// TwinCAT 3 PLC project Lectures
// ProgramVersion: 3.1.4024.0
// libraries:
//   Tc2_Standard, * (Beckhoff Automation GmbH)
//   Tc2_System, * (Beckhoff Automation GmbH)
//   Tc3_Module, * (Beckhoff Automation GmbH)
// project tree:
//   DUTs/ Item.TcDUT, Location.TcDUT (not stored)
//   GVLs/ Automatic.TcGVL, IO.TcGVL (not stored)
//   / PlcTask.TcTTO (not stored)
//   POUs/ AutomaticControl.TcPOU, CountCurrentPosition1.TcPOU, Initialize.TcPOU (not stored), ManualControl.TcPOU, MAIN.TcPOU, MotorSelection.TcPOU, Recipe1.TcPOU, Recipe11.TcPOU, Recipe2.TcPOU, RestorePreviousAutomaticState.TcPOU, Safety1.TcPOU
//   POUs/Lectures%27 programs/ p00_true_false.TcPOU (not stored), p01_sequential.TcPOU (not stored), p02_clock.TcPOU (not stored), p03_SR1.TcPOU (not stored), p04_latch.TcPOU (not stored), p05_posEdge.TcPOU (not stored), p06_frontDetection.TcPOU (not stored), p07_memoryCell.TcPOU (not stored), p08_counter.TcPOU (not stored), p09_timers.TcPOU (not stored), p10_directionalInterlock.TcPOU (not stored), p11_logicalFunction.TcPOU (not stored), p12_controlLight.TcPOU (not stored)
// real-time tasks:
//   TASK PlcTask1: cycle T#10ms, priority 21, ADS port 351
//   TASK PlcTask: cycle T#10ms, priority 20, ADS port 350
// I/O:
//   DEVICE Device 1 (EtherCAT), AmsNetId 172.31.192.1.2.1
//     Term 1 (EK1200) [EK1200-7000 EtherCAT Power supply (1,5A E-Bus)]
//       Term 2 (EL1859) [EL1859 8Ch. Dig. Input 24V, 3ms, 8Ch. Dig. Output 24V, 0.5A]
//       Term 3 (EL1859) [EL1859 8Ch. Dig. Input 24V, 3ms, 8Ch. Dig. Output 24V, 0.5A]
//       Term 4 (EL9011) [EL9011 End Terminal]
//   DEVICE Device 2 (NOV-DP-RAM) (disabled)
//   DEVICE Device 3 (CX7000), AmsNetId 172.31.192.1.4.1
//     Term 1 (CX7028) [CX7028-0000-0121]
//       modules: Module 1 (DIO_2x), Module 2 (Empty Module), Module 3 (DIO_2x), Module 4 (Empty Module), Module 5 (DI_2x), Module 6 (Empty Module), Module 7 (DI_2x), Module 8 (Empty Module)
// variable links:
//   Lectures/Lectures Instance <-> Device 1 (EtherCAT)/Term 1 (EK1200)/Term 2 (EL1859)
//     PlcTask Inputs/IO.EndExtensionSensor <-> Channel 3/Input
//     PlcTask Inputs/IO.EndGripSensor <-> Channel 7/Input
//     PlcTask Inputs/IO.EndLiftingSensor <-> Channel 5/Input
//     PlcTask Inputs/IO.EndRotationSensor <-> Channel 1/Input
//     PlcTask Inputs/IO.StepExtensionSwitch <-> Channel 4/Input
//     PlcTask Inputs/IO.StepGripSwitch <-> Channel 8/Input
//     PlcTask Inputs/IO.StepLiftingSwitch <-> Channel 6/Input
//     PlcTask Inputs/IO.StepRotatonSwitch <-> Channel 2/Input
//     PlcTask Outputs/IO.MotorExtension <-> Channel 12/Output
//     PlcTask Outputs/IO.MotorExtensionDirection <-> Channel 11/Output
//     PlcTask Outputs/IO.MotorGrip <-> Channel 16/Output
//     PlcTask Outputs/IO.MotorGripDirection <-> Channel 15/Output
//     PlcTask Outputs/IO.MotorLifting <-> Channel 14/Output
//     PlcTask Outputs/IO.MotorLiftingDirection <-> Channel 13/Output
//     PlcTask Outputs/IO.MotorRotation <-> Channel 10/Output
//     PlcTask Outputs/IO.MotorRotationDirection <-> Channel 9/Output
//   Lectures/Lectures Instance <-> Device 3 (CX7000)/Term 1 (CX7028)
//     PlcTask Inputs/IO.ButtonGreen <-> Module 3 (DIO_2x)/DIO_2x Input Channel 2/Input
//     PlcTask Inputs/IO.ButtonLowerLeft <-> Module 5 (DI_2x)/DI_2x Input Channel 1/Input
//     PlcTask Inputs/IO.ButtonLowerRight <-> Module 5 (DI_2x)/DI_2x Input Channel 2/Input
//     PlcTask Inputs/IO.ButtonRed <-> Module 1 (DIO_2x)/DIO_2x Input Channel 1/Input
//     PlcTask Inputs/IO.ButtonUpperLeft <-> Module 1 (DIO_2x)/DIO_2x Input Channel 2/Input
//     PlcTask Inputs/IO.ButtonUpperRight <-> Module 3 (DIO_2x)/DIO_2x Input Channel 1/Input
//     PlcTask Inputs/IO.Switch <-> Module 7 (DI_2x)/DI_2x Input Channel 1/Input
//     PlcTask Outputs/IO.LEDBlueLower <-> Module 3 (DIO_2x)/DIO_2x Output Channel 2/Output
//     PlcTask Outputs/IO.LEDBlueUpper <-> Module 1 (DIO_2x)/DIO_2x Output Channel 2/Output
//     PlcTask Outputs/IO.LEDGreen <-> Module 3 (DIO_2x)/DIO_2x Output Channel 1/Output
//     PlcTask Outputs/IO.LEDRed <-> Module 1 (DIO_2x)/DIO_2x Output Channel 1/Output

// ---- DUTs/Item.TcDUT
TYPE Item :
STRUCT
END_STRUCT
END_TYPE

// ---- GVLs/Automatic.TcGVL
{attribute 'qualified_only'}
VAR_GLOBAL
	RCurrentlyMoving: BOOL;
	RotationPositionAuto: INT;
	RotationPositionCurrent: INT;
	SafetyRON: BOOL;
	
	LCurrentlyMoving: BOOL;
	LiftingPositionAuto: INT;
	LiftingPositionCurrent: INT;
	SafetyLON: BOOL;
	
	ECurrentlyMoving: BOOL;
	ExtensionPositionAuto: INT;
	ExtensionPositionCurrent: INT;
	SafetyEON: BOOL;
	
	GCurrentlyMoving: BOOL;
	GripPositionAuto: INT;
	GripPositionCurrent: INT;
	SafetyGON: BOOL;
	
	AllRestored: BOOL;
END_VAR

// ---- POUs/AutomaticControl.TcPOU
FUNCTION_BLOCK PUBLIC AutomaticControl
VAR_INPUT
    Switch: BOOL;
END_VAR
VAR
    State: INT := 0;
    ExecutingRecipe1: BOOL := FALSE;
    ExecutingRecipe2: BOOL := FALSE;
	myRecipe1: Recipe1;
    myRecipe2: Recipe2;
    Tmp: BOOL;
    RestorePreviousAutomaticState: RestorePreviousAutomaticState;
	CountCurrentPosition1: CountCurrentPosition1;
	Safety: Safety1;
END_VAR
VAR_OUTPUT
    Output: BOOL := TRUE;
END_VAR

// TwinCAT ensures that all POUs, including your AutomaticControl program 
// and Recipe1() Function Block, are executed once per cycle.

// for debugging purposes:
IF IO.ButtonRed THEN
	IO.Initialized := FALSE;
END_IF


IF (NOT IO.Initialized) THEN
	Initialize();
ELSIF (NOT IO.Switch) AND IO.PreviousManualMode THEN
	CountCurrentPosition1();
	Safety();
	RestorePreviousAutomaticState();
ELSE
	CountCurrentPosition1();
	Safety();
	
    IF (IO.ButtonUpperLeft OR ExecutingRecipe1) AND Automatic.AllRestored THEN
        //ExecutingRecipe1 := TRUE;
		//Recipe11();
        //ExecutingRecipe1 := NOT Recipe11.SuccesfullyEnded; // Update ExecutingRecipe1 based on output
		myRecipe1.ExecutingRecipe1 := TRUE;
		ExecutingRecipe1 := NOT myRecipe1.SuccesfullyEnded;
    ELSIF (NOT ExecutingRecipe1) AND (IO.ButtonUpperRight OR ExecutingRecipe2) AND Automatic.AllRestored THEN
        ExecutingRecipe2 := TRUE;
        myRecipe2.ExecutingRecipe2 := ExecutingRecipe2; // Pass input to the function block
        //myRecipe2(); // Call the function block
        ExecutingRecipe2 := NOT myRecipe2.SuccesfullyEnded; // Update ExecutingRecipe2 based on output
    END_IF
END_IF




RETURN;

END_FUNCTION_BLOCK

// ---- POUs/Recipe1.TcPOU
FUNCTION_BLOCK Recipe1
VAR_INPUT
	ExecutingRecipe1: BOOL;
END_VAR
VAR_OUTPUT
	SuccesfullyEnded: BOOL := FALSE;
END_VAR
VAR
	State: INT := 0;
	WoodInitialLiftingPosition: INT := 50;
	InitialExtensionPosition: INT := 388;
	MaxGripPosition: INT := 150;
	RotationDropOffPosition: INT := 300;
	PlasticsInitialLiftingPosition: INT := 250;
	PlasticsDropOffExtensionPosition: INT := 300;
	MetalInitialLiftingPosition: INT := 400;
	MetalDropOffExtensionPosition: INT := 500;
END_VAR

IF ExecutingRecipe1 THEN	// we start executing recipe1 (again)
	SuccesfullyEnded := FALSE;
END_IF

IF (NOT IO.Switch) AND (NOT SuccesfullyEnded) THEN
	IO.LEDGreen := 1;
	// WOOD:
	IF State = 0 THEN
		IF Automatic.LiftingPositionAuto < WoodInitialLiftingPosition THEN
			IO.MotorLiftingDirection := 0;
			IF (NOT Automatic.SafetyLON) THEN
				Automatic.LCurrentlyMoving := TRUE;
				IO.MotorLifting := 1;
			END_IF
		ELSE
			State := 1;
			IO.MotorLifting := 0;
			Automatic.LCurrentlyMoving := FALSE;
		END_IF
	ELSIF State = 1 THEN
		IF Automatic.ExtensionPositionAuto < InitialExtensionPosition THEN
			IO.MotorExtensionDirection := 0;
			IF NOT Automatic.SafetyEON THEN
				Automatic.ECurrentlyMoving := TRUE;
				IO.MotorExtension := 1;
			END_IF
		ELSE
			State := 2;
			IO.MotorExtension := 0;
			Automatic.ECurrentlyMoving := FALSE;
		END_IF
	ELSIF State = 2 THEN
		IF Automatic.GripPositionAuto < MaxGripPosition THEN
			IO.MotorGripDirection := 0;
			IF NOT Automatic.SafetyGON THEN
				Automatic.GCurrentlyMoving := TRUE;
				IO.MotorGrip := 1;
			END_IF
		ELSE
			State := 3;
			IO.MotorGrip := 0;
			Automatic.GCurrentlyMoving := FALSE;
		END_IF
	ELSIF State = 3 THEN
		IF NOT IO.EndLiftingSensor THEN
			IO.MotorLiftingDirection := 1;
			IF NOT Automatic.SafetyLON THEN
				Automatic.GCurrentlyMoving := TRUE;
				IO.MotorLifting := 1;
			END_IF
		ELSE
			State := 4;
			IO.MotorLifting := 0;
			Automatic.LCurrentlyMoving := FALSE;
		END_IF
	ELSIF State = 4 THEN
		IF Automatic.RotationPositionAuto < RotationDropOffPosition THEN
			IO.MotorRotationDirection := 0;
			IF NOT Automatic.SafetyRON THEN
				Automatic.RCurrentlyMoving := TRUE;
				IO.MotorRotation := 1;
			END_IF
		ELSE
			State := 5;
			IO.MotorRotation := 0;
			Automatic.RCurrentlyMoving := FALSE;
		END_IF
	ELSIF State = 5 THEN
		IF NOT IO.EndExtensionSensor THEN	// it drops wood in the nearest bin
			IO.MotorExtensionDirection := 1;
			IF NOT Automatic.SafetyEON THEN
				Automatic.ECurrentlyMoving := TRUE;
				IO.MotorExtension := 1;
			END_IF
		ELSE
			State := 6;
			IO.MotorExtension := 0;
			Automatic.ECurrentlyMoving := FALSE;
		END_IF
	ELSIF State = 6 THEN
		IF NOT IO.EndGripSensor THEN
			IO.MotorGripDirection := 1;
			IF NOT Automatic.SafetyGON THEN
				Automatic.GCurrentlyMoving := TRUE;
				IO.MotorGrip := 1;
			END_IF
		ELSE
			State := 7;
			IO.MotorGrip := 0;
			Automatic.GCurrentlyMoving := FALSE;
		END_IF
	ELSIF State = 7 THEN
		IF NOT IO.EndRotationSensor THEN
			IO.MotorRotationDirection := 1;
			IF NOT Automatic.SafetyRON THEN
				Automatic.RCurrentlyMoving := TRUE;
				IO.MotorRotation := 1;
			END_IF
		ELSE
			State := 8;
			IO.MotorRotation := 0;
			Automatic.RCurrentlyMoving := FALSE;
		END_IF
	END_IF
	
	// PLASTICS:
	IF State = 8 THEN
		IF Automatic.LiftingPositionAuto < PlasticsInitialLiftingPosition THEN
			IO.MotorLiftingDirection := 0;
			IF NOT Automatic.SafetyLON THEN
				Automatic.LCurrentlyMoving := TRUE;
				IO.MotorLifting := 1;
			END_IF
		ELSE
			State := 9;
			IO.MotorLifting := 0;
			Automatic.LCurrentlyMoving := FALSE;
		END_IF
	ELSIF State = 9 THEN
		IF Automatic.ExtensionPositionAuto < InitialExtensionPosition THEN
			IO.MotorExtensionDirection := 0;
			IF NOT Automatic.SafetyEON THEN
				Automatic.ECurrentlyMoving := TRUE;
				IO.MotorExtension := 1;
			END_IF
		ELSE
			State := 10;
			IO.MotorExtension := 0;
			Automatic.ECurrentlyMoving := FALSE;
		END_IF
	ELSIF State = 10 THEN
		IF Automatic.GripPositionAuto < MaxGripPosition THEN
			IO.MotorGripDirection := 0;
			IF NOT Automatic.SafetyGON THEN
				Automatic.GCurrentlyMoving := TRUE;
				IO.MotorGrip := 1;
			END_IF
		ELSE
			State := 11;
			IO.MotorGrip := 0;
			Automatic.GCurrentlyMoving := FALSE;
		END_IF
	ELSIF State = 11 THEN
		IF NOT IO.EndLiftingSensor THEN
			IO.MotorLiftingDirection := 1;
			IF NOT Automatic.SafetyLON THEN
				Automatic.LCurrentlyMoving := TRUE;
				IO.MotorLifting := 1;
			END_IF
		ELSE
			State := 12;
			IO.MotorLifting := 0;
			Automatic.LCurrentlyMoving := FALSE;
		END_IF
	ELSIF State = 12 THEN
		IF Automatic.RotationPositionAuto < RotationDropOffPosition THEN
			IO.MotorRotationDirection := 0;
			IF NOT Automatic.SafetyRON THEN
				Automatic.RCurrentlyMoving := TRUE;
				IO.MotorRotation := 1;
			END_IF
		ELSE
			State := 13;
			IO.MotorRotation := 0;
			Automatic.RCurrentlyMoving := FALSE;
		END_IF
	ELSIF State = 13 THEN
		IF Automatic.ExtensionPositionAuto > PlasticsDropOffExtensionPosition THEN	// it drops plastics into second nearest bin
			IO.MotorExtensionDirection := 1;
			IF NOT Automatic.SafetyEON THEN
				Automatic.ECurrentlyMoving := TRUE;
				IO.MotorExtension := 1;
			END_IF
		ELSE
			State := 14;
			IO.MotorExtension := 0;
			Automatic.ECurrentlyMoving := FALSE;
		END_IF
	ELSIF State = 14 THEN
		IF NOT IO.EndGripSensor THEN
			IO.MotorGripDirection := 1;
			IF NOT Automatic.SafetyGON THEN
				Automatic.GCurrentlyMoving := TRUE;
				IO.MotorGrip := 1;
			END_IF
		ELSE
			State := 15;
			IO.MotorGrip := 0;
			Automatic.GCurrentlyMoving := FALSE;
		END_IF
	ELSIF State = 15 THEN
		IF NOT IO.EndRotationSensor THEN
			IO.MotorRotationDirection := 0;
			IF NOT Automatic.SafetyRON THEN
				Automatic.RCurrentlyMoving := TRUE;
				IO.MotorRotation := 1;
			END_IF
		ELSE
			State := 16;
			IO.MotorRotation := 0;
			Automatic.RCurrentlyMoving := FALSE;
		END_IF
	END_IF
	
	// METAL:
	IF State = 16 THEN
		IF Automatic.LiftingPositionAuto < MetalInitialLiftingPosition THEN
			IO.MotorLiftingDirection := 0;
			IF NOT Automatic.SafetyLON THEN
				Automatic.LCurrentlyMoving := TRUE;
				IO.MotorLifting := 1;
			END_IF
		ELSE
			State := 17;
			IO.MotorLifting := 0;
			Automatic.LCurrentlyMoving := FALSE;
		END_IF
	ELSIF State = 17 THEN
		IF Automatic.ExtensionPositionAuto < InitialExtensionPosition THEN
			IO.MotorExtensionDirection := 0;
			IF NOT Automatic.SafetyEON THEN
				Automatic.ECurrentlyMoving := TRUE;
				IO.MotorExtension := 1;
			END_IF
		ELSE
			State := 18;
			IO.MotorExtension := 0;
			Automatic.ECurrentlyMoving := FALSE;
		END_IF
	ELSIF State = 18 THEN
		IF Automatic.GripPositionAuto < MaxGripPosition THEN
			IO.MotorGripDirection := 0;
			IF NOT Automatic.SafetyGON THEN
				Automatic.GCurrentlyMoving := TRUE;
				IO.MotorGrip := 1;
			END_IF
		ELSE
			State := 19;
			IO.MotorGrip := 0;
			Automatic.GCurrentlyMoving := FALSE;
		END_IF
	ELSIF State = 19 THEN
		IF NOT IO.EndLiftingSensor THEN
			IO.MotorLiftingDirection := 1;
			IF NOT Automatic.SafetyLON THEN
				Automatic.LCurrentlyMoving := TRUE;
				IO.MotorLifting := 1;
			END_IF
		ELSE
			State := 20;
			IO.MotorLifting := 0;
			Automatic.LCurrentlyMoving := FALSE;
		END_IF
	ELSIF State = 20 THEN
		IF Automatic.RotationPositionAuto < RotationDropOffPosition THEN
			IO.MotorRotationDirection := 0;
			IF NOT Automatic.SafetyRON THEN
				Automatic.RCurrentlyMoving := TRUE;
				IO.MotorRotation := 1;
			END_IF
		ELSE
			State := 21;
			IO.MotorRotation := 0;
			Automatic.RCurrentlyMoving := FALSE;
		END_IF
	ELSIF State = 21 THEN
		IF Automatic.ExtensionPositionAuto > MetalDropOffExtensionPosition THEN	// it drops metal into farthest bin
			IO.MotorExtensionDirection := 1;
			IF NOT Automatic.SafetyEON THEN
				Automatic.ECurrentlyMoving := TRUE;
				IO.MotorExtension := 1;
			END_IF
		ELSE
			State := 22;
			IO.MotorExtension := 0;
			Automatic.ECurrentlyMoving := FALSE;
		END_IF
	ELSIF State = 22 THEN
		IF NOT IO.EndGripSensor THEN
			IO.MotorGripDirection := 1;
			IF NOT Automatic.SafetyGON THEN
				Automatic.GCurrentlyMoving := TRUE;
				IO.MotorGrip := 1;
			END_IF
		ELSE
			State := 23;
			IO.MotorGrip := 0;
			Automatic.GCurrentlyMoving := FALSE;
		END_IF
	ELSIF State = 23 THEN
		IF NOT IO.EndRotationSensor THEN
			IO.MotorRotationDirection := 1;
			IF NOT Automatic.SafetyRON THEN
				Automatic.RCurrentlyMoving := TRUE;
				IO.MotorRotation := 1;
			END_IF
		ELSE
			State := 24;
			IO.MotorRotation := 0;
			Automatic.RCurrentlyMoving := FALSE;
		END_IF
	ELSIF State = 24 THEN
		SuccesfullyEnded := TRUE;
		State := 0;
		RETURN;
	END_IF
END_IF
RETURN;

END_FUNCTION_BLOCK

// ---- POUs/Recipe2.TcPOU
FUNCTION_BLOCK PUBLIC Recipe2
VAR_INPUT
	ExecutingRecipe2: BOOL;
END_VAR
VAR_OUTPUT
	SuccesfullyEnded: BOOL := FALSE;
END_VAR
VAR
	State: INT := 0;
	InitialRotationPosition: INT := 140;
	InitialLiftingPosition: INT := 200;
	MaxGripPosition: INT := 160;
END_VAR

// Recipe is sequence of moves to execute the task.

IF ExecutingRecipe2 THEN	// we start executing recipe2 (again)
	SuccesfullyEnded := FALSE;
END_IF

IF NOT IO.Switch AND NOT SuccesfullyEnded THEN
	// WOOD:
	IF State = 0 THEN
		IF Automatic.RotationPositionAuto < InitialRotationPosition THEN
			IO.MotorRotationDirection := 0;
			IF NOT Automatic.SafetyRON THEN
				Automatic.RCurrentlyMoving := TRUE;
				IO.MotorRotation := 1;
			END_IF
		ELSE
			State := 1;
			IO.MotorRotation := 0;
			Automatic.RCurrentlyMoving := FALSE;
		END_IF
	ELSIF State = 1 THEN
		IF Automatic.LiftingPositionAuto < InitialLiftingPosition THEN
			IO.MotorLiftingDirection := 1;
			IF NOT Automatic.SafetyLON THEN
				Automatic.LCurrentlyMoving := TRUE;
				IO.MotorLifting := 1;
			END_IF
		ELSE
			State := 2;
			IO.MotorLifting := 0;
			Automatic.LCurrentlyMoving := FALSE;
		END_IF
	ELSIF State = 2 THEN
		IF Automatic.GripPositionAuto < MaxGripPosition THEN
			IO.MotorGripDirection := 0;
			IF NOT Automatic.SafetyGON THEN
				Automatic.GCurrentlyMoving := TRUE;
				IO.MotorGrip := 1;
			END_IF
		ELSE
			State := 3;
			IO.MotorGrip := 0;
			Automatic.GCurrentlyMoving := FALSE;
		END_IF
	ELSIF State = 3 THEN
		IF NOT IO.EndLiftingSensor THEN
			IO.MotorLiftingDirection := 0;
			IF NOT Automatic.SafetyLON THEN
				Automatic.GCurrentlyMoving := TRUE;
				IO.MotorLifting := 1;
			END_IF
		ELSE
			State := 4;
			IO.MotorLifting := 0;
			Automatic.GCurrentlyMoving := FALSE;
		END_IF
	ELSIF State = 4 THEN
		IF NOT IO.EndRotationSensor THEN
			IO.MotorRotationDirection := 1;
			IF NOT Automatic.SafetyRON THEN
				Automatic.RCurrentlyMoving := TRUE;
				IO.MotorRotation := 1;
			END_IF
		ELSE
			State := 5;
			IO.MotorRotation := 0;
			Automatic.RCurrentlyMoving := FALSE;
		END_IF
	ELSIF State = 5 THEN
		IF NOT IO.EndGripSensor THEN		// it places the cylinder onto the platform
			IO.MotorGripDirection := 1;
			IF NOT Automatic.SafetyGON THEN
				Automatic.GCurrentlyMoving := TRUE;
				IO.MotorGrip := 1;
			END_IF
		ELSE
			State := 6;
			IO.MotorGrip := 0;
			Automatic.GCurrentlyMoving := FALSE;
		END_IF
	ELSIF State = 6 THEN
		SuccesfullyEnded := TRUE;
		State := 0;
		RETURN;
	END_IF
END_IF

END_FUNCTION_BLOCK

// ---- POUs/RestorePreviousAutomaticState.TcPOU
FUNCTION_BLOCK PUBLIC RestorePreviousAutomaticState
VAR_INPUT
END_VAR
VAR_OUTPUT
END_VAR
VAR
	RotationRestored: BOOL := FALSE;
	LiftingRestored: BOOL := FALSE;
	ExtensionRestored: BOOL := FALSE;
	GripRestored: BOOL := FALSE;
END_VAR

IF IO.PreviousManualMode THEN
	Automatic.AllRestored := FALSE;
END_IF

// reset rotation:
IF Automatic.RotationPositionAuto - Automatic.RotationPositionCurrent > 5 AND (NOT RotationRestored) AND (NOT Automatic.SafetyRON) THEN
	IO.MotorRotationDirection := 0;
	Automatic.RCurrentlyMoving := TRUE;
	IO.MotorRotation := 1;
ELSIF Automatic.RotationPositionCurrent - Automatic.RotationPositionAuto > 5 AND (NOT RotationRestored) AND (NOT Automatic.SafetyRON) THEN
	IO.MotorRotationDirection := 1;
	Automatic.RCurrentlyMoving := TRUE;
	IO.MotorRotation := 1;
ELSE
	Automatic.RCurrentlyMoving := FALSE;
	IO.MotorRotation := 0;
	RotationRestored := TRUE;
END_IF

// reset lifting:
IF Automatic.LiftingPositionAuto - Automatic.LiftingPositionCurrent > 5 AND (NOT LiftingRestored) AND (NOT Automatic.SafetyLON) THEN
	IO.MotorLiftingDirection := 0;
	Automatic.LCurrentlyMoving := TRUE;
	IO.MotorLifting := 1;
ELSIF Automatic.LiftingPositionCurrent - Automatic.LiftingPositionAuto > 5 AND (NOT LiftingRestored) AND (NOT Automatic.SafetyLON) THEN
	IO.MotorLiftingDirection := 0;
	Automatic.LCurrentlyMoving := TRUE;
	IO.MotorLifting := 1;
ELSE
	Automatic.LCurrentlyMoving := FALSE;
	IO.MotorLifting := 0;
	LiftingRestored := TRUE;
END_IF

// reset extension:
IF Automatic.ExtensionPositionAuto - Automatic.ExtensionPositionCurrent > 5 AND (NOT ExtensionRestored) AND (NOT Automatic.SafetyEON) THEN
	IO.MotorExtensionDirection := 0;
	Automatic.ECurrentlyMoving := TRUE;
	IO.MotorExtension := 1;
ELSIF Automatic.ExtensionPositionCurrent - Automatic.ExtensionPositionAuto > 5 AND (NOT ExtensionRestored) AND (NOT Automatic.SafetyEON) THEN
	IO.MotorExtensionDirection := 0;
	Automatic.ECurrentlyMoving := TRUE;
	IO.MotorExtension := 1;
ELSE
	Automatic.ECurrentlyMoving := FALSE;
	IO.MotorExtension := 0;
	ExtensionRestored := TRUE;
END_IF

// reset grip:
IF Automatic.GripPositionAuto - Automatic.GripPositionCurrent > 5 AND (NOT GripRestored) AND (NOT Automatic.SafetyGON) THEN
	IO.MotorGripDirection := 0;
	Automatic.GCurrentlyMoving := TRUE;
	IO.MotorGrip := 1;
ELSIF Automatic.GripPositionCurrent - Automatic.GripPositionAuto > 5 AND (NOT GripRestored) AND (NOT Automatic.SafetyGON) THEN
	IO.MotorGripDirection := 0;
	Automatic.GCurrentlyMoving := TRUE;
	IO.MotorGrip := 1;
ELSE
	Automatic.GCurrentlyMoving := FALSE;
	IO.MotorGrip := 0;
	GripRestored := TRUE;
END_IF

// if all restored then go on to exeecute recipes in AutomaticControl:
IF RotationRestored AND LiftingRestored AND ExtensionRestored AND GripRestored THEN
	IO.PreviousManualMode := FALSE;
	Automatic.AllRestored := TRUE;
	
	RotationRestored := FALSE;
	ExtensionRestored := FALSE;
	LiftingRestored := FALSE;
	GripRestored := FALSE;
	Automatic.RCurrentlyMoving := FALSE;
	Automatic.ECurrentlyMoving := FALSE;
	Automatic.LCurrentlyMoving := FALSE;
	Automatic.GCurrentlyMoving := FALSE;
END_IF

END_FUNCTION_BLOCK

// ---- POUs/CountCurrentPosition1.TcPOU
FUNCTION_BLOCK CountCurrentPosition1
VAR_INPUT
END_VAR
VAR_OUTPUT
END_VAR
VAR
END_VAR

IF IO.Initialized THEN
	
	// COUNT ROTATION:
	IF IO.StepRotatonSwitch = 1 AND Automatic.RCurrentlyMoving THEN
		// away from the sensor:
		IF IO.MotorRotationDirection = 0 THEN
			IF (NOT IO.Switch) THEN		// in automatic mode
				IF IO.PreviousManualMode THEN	
					Automatic.RotationPositionCurrent := Automatic.RotationPositionCurrent + 1;
				ELSE	// to restore the state
					Automatic.RotationPositionCurrent := Automatic.RotationPositionCurrent + 1;
					Automatic.RotationPositionAuto := Automatic.RotationPositionAuto + 1;
				END_IF
			ELSE		// in manual mode
				Automatic.RotationPositionCurrent := Automatic.RotationPositionCurrent + 1;
			END_IF
		// towards the sensor:
		ELSE
			IF (NOT IO.Switch) THEN		// in automatic mode
				IF IO.PreviousManualMode THEN	
					Automatic.RotationPositionCurrent := Automatic.RotationPositionCurrent - 1;
				ELSE	// to restore the state
					Automatic.RotationPositionCurrent := Automatic.RotationPositionCurrent - 1;
					Automatic.RotationPositionAuto := Automatic.RotationPositionAuto - 1;
				END_IF
			ELSE		// in manual mode
				Automatic.RotationPositionCurrent := Automatic.RotationPositionCurrent - 1;
			END_IF
		END_IF
	END_IF
	
	// COUNT Extension: (-------edino še NESPREMENJENO--------)
	IF IO.StepExtensionSwitch = 1 THEN
		IF IO.MotorExtensionDirection = 0 THEN
			IF (NOT IO.Switch) AND Automatic.ECurrentlyMoving THEN
				IF IO.PreviousManualMode THEN
					Automatic.ExtensionPositionCurrent := Automatic.ExtensionPositionCurrent + 1;
				ELSE
					Automatic.ExtensionPositionAuto := Automatic.ExtensionPositionAuto + 1;
					Automatic.ExtensionPositionCurrent := Automatic.ExtensionPositionCurrent + 1;
				END_IF
			ELSIF Automatic.ECurrentlyMoving THEN
				Automatic.ExtensionPositionCurrent := Automatic.ExtensionPositionCurrent + 1;
			END_IF
		ELSE
			IF (NOT IO.Switch) AND Automatic.ECurrentlyMoving THEN
				IF IO.PreviousManualMode THEN
					Automatic.ExtensionPositionCurrent := Automatic.ExtensionPositionCurrent - 1;
				ELSE
					Automatic.ExtensionPositionAuto := Automatic.ExtensionPositionAuto - 1;
					Automatic.ExtensionPositionCurrent := Automatic.ExtensionPositionCurrent - 1;
				END_IF
			ELSIF Automatic.ECurrentlyMoving THEN
				Automatic.ExtensionPositionCurrent := Automatic.ExtensionPositionCurrent - 1;
			END_IF
		END_IF
	END_IF
	
	// COUNT Lifting:
	IF IO.StepLiftingSwitch = 1 AND Automatic.LCurrentlyMoving THEN
		// away from the sensor:
		IF IO.MotorLiftingDirection = 0 THEN
			IF (NOT IO.Switch) THEN		// in automatic mode
				IF IO.PreviousManualMode THEN
					Automatic.LiftingPositionCurrent := Automatic.LiftingPositionCurrent + 1;
				ELSE	// to restore the state
					Automatic.LiftingPositionCurrent := Automatic.LiftingPositionCurrent + 1;
					Automatic.LiftingPositionAuto := Automatic.LiftingPositionAuto + 1;
				END_IF
			ELSE		// in manual mode
				Automatic.LiftingPositionCurrent := Automatic.LiftingPositionCurrent + 1;
			END_IF
		// towards the sensor:
		ELSE
			IF (NOT IO.Switch) THEN		// in automatic mode
				IF IO.PreviousManualMode THEN
					Automatic.LiftingPositionCurrent := Automatic.LiftingPositionCurrent - 1;
				ELSE	// to restore the state
					Automatic.LiftingPositionAuto := Automatic.LiftingPositionAuto - 1;
					Automatic.LiftingPositionCurrent := Automatic.LiftingPositionCurrent - 1;
				END_IF
			ELSE		// in manual mode
				Automatic.LiftingPositionCurrent := Automatic.LiftingPositionCurrent - 1;
			END_IF
		END_IF
	END_IF
	
	// COUNT Grip:
	IF IO.StepGripSwitch = 1 AND Automatic.GCurrentlyMoving THEN
		IF IO.MotorGripDirection = 0 THEN
			IF (NOT IO.Switch) THEN		// in automatic mode
				IF IO.PreviousManualMode THEN
					Automatic.GripPositionCurrent := Automatic.GripPositionCurrent + 1;
				ELSE
					Automatic.GripPositionAuto := Automatic.GripPositionAuto + 1;
					Automatic.GripPositionCurrent := Automatic.GripPositionCurrent + 1;
				END_IF
			ELSE		// in manual mode
				Automatic.GripPositionCurrent := Automatic.GripPositionCurrent + 1;
			END_IF
		ELSE
			IF (NOT IO.Switch) THEN		// in automatic mode
				IF IO.PreviousManualMode THEN
					Automatic.GripPositionCurrent := Automatic.GripPositionCurrent - 1;
				ELSE
					Automatic.GripPositionAuto := Automatic.GripPositionAuto - 1;
					Automatic.GripPositionCurrent := Automatic.GripPositionCurrent - 1;
				END_IF
			ELSE		// in manual mode
				Automatic.GripPositionCurrent := Automatic.GripPositionCurrent - 1;
			END_IF
		END_IF
	END_IF
	
END_IF

END_FUNCTION_BLOCK

// ---- POUs/Safety1.TcPOU
FUNCTION_BLOCK Safety1
VAR_INPUT
END_VAR
VAR_OUTPUT
END_VAR
VAR
	MaxRotationPosition: INT := 555;
	MaxLiftingPosition: INT := 270;
	MaxExtensionPosition: INT := 445;
	MaxGripPosition: INT := 155;
END_VAR

// Safety for Rotation:
IF Automatic.RotationPositionCurrent >= MaxRotationPosition AND NOT IO.ButtonLowerLeft AND NOT IO.MotorRotationDirection = 1 THEN
	Automatic.SafetyRON := TRUE;
	IO.MotorRotation := 0;
	IF Automatic.RotationPositionCurrent >= MaxRotationPosition THEN
		Automatic.RotationPositionCurrent := MaxRotationPosition;
	END_IF
	//Automatic.MotorR.CurrentlyMoving := FALSE;
	Automatic.RCurrentlyMoving := FALSE;
END_IF
IF IO.MotorRotationDirection = 0 THEN
	Automatic.SafetyRON := FALSE;
END_IF
IF IO.EndRotationSensor THEN
	IF IO.MotorRotationDirection = 0 THEN
		Automatic.SafetyRON := FALSE;
	ELSE
		Automatic.SafetyRON := TRUE;
		Automatic.RotationPositionCurrent := 0;
		//Automatic.MotorR.CurrentlyMoving := FALSE;
		Automatic.RCurrentlyMoving := FALSE;
	END_IF
END_IF

// Safety for Lifting:
IF Automatic.LiftingPositionCurrent >= MaxLiftingPosition AND NOT IO.ButtonLowerLeft AND NOT IO.MotorLiftingDirection = 1 THEN
	Automatic.SafetyLON := TRUE;
	IO.MotorLifting := 0;
	IF Automatic.LiftingPositionCurrent >= MaxLiftingPosition THEN
		Automatic.LiftingPositionCurrent := MaxLiftingPosition;
	END_IF
	//Automatic.MotorL.CurrentlyMoving := FALSE;
	Automatic.LCurrentlyMoving := FALSE;
END_IF
IF IO.MotorLiftingDirection = 0 THEN
	Automatic.SafetyLON := FALSE;
END_IF
IF IO.EndLiftingSensor THEN
	IF IO.MotorLiftingDirection = 0 THEN
		Automatic.SafetyLON := FALSE;
	ELSE
		Automatic.SafetyLON := TRUE;
		Automatic.LiftingPositionCurrent := 0;
		//Automatic.MotorL.CurrentlyMoving := FALSE;
		Automatic.RCurrentlyMoving := FALSE;
	END_IF
END_IF

// Safety for Extension:
IF Automatic.ExtensionPositionCurrent >= MaxExtensionPosition AND NOT IO.ButtonLowerLeft AND NOT IO.MotorExtensionDirection = 1 THEN
	Automatic.SafetyEON := TRUE;
	IO.MotorExtension := 0;
	IF Automatic.ExtensionPositionCurrent >= MaxExtensionPosition THEN
		Automatic.ExtensionPositionCurrent := MaxExtensionPosition;
	END_IF
	//Automatic.MotorE.CurrentlyMoving := FALSE;
	Automatic.ECurrentlyMoving := FALSE;
END_IF
IF IO.MotorExtensionDirection = 0 THEN
	Automatic.SafetyEON := FALSE;
END_IF
IF IO.EndExtensionSensor THEN
	IF IO.MotorExtensionDirection = 0 THEN
		Automatic.SafetyEON := FALSE;
	ELSE
		Automatic.SafetyEON := TRUE;
		Automatic.ExtensionPositionCurrent := 0;
		//Automatic.MotorE.CurrentlyMoving := FALSE;
		Automatic.ECurrentlyMoving := FALSE;
	END_IF
END_IF

// Safety for Grip:
IF Automatic.GripPositionCurrent >= MaxGripPosition AND NOT IO.ButtonLowerLeft AND IO.MotorGripDirection = 0 THEN
	Automatic.SafetyGON := TRUE;
	IO.MotorGrip := 0;
	IF Automatic.GripPositionCurrent >= MaxGripPosition THEN
		Automatic.GripPositionCurrent := MaxGripPosition;
	END_IF
	//Automatic.GCurrentlyMoving := FALSE;
	Automatic.GCurrentlyMoving := FALSE;
END_IF
IF IO.MotorGripDirection = 1 THEN
	Automatic.SafetyGON := FALSE;
END_IF
IF IO.EndGripSensor THEN
	IF IO.MotorGripDirection = 0 THEN
		Automatic.SafetyGON := FALSE;
	ELSE
		Automatic.SafetyGON := TRUE;
		Automatic.GripPositionCurrent := 0;
		//Automatic.GCurrentlyMoving := FALSE;
		Automatic.GCurrentlyMoving := FALSE;
	END_IF
END_IF

END_FUNCTION_BLOCK

// ---- POUs/ManualControl.TcPOU
FUNCTION_BLOCK PUBLIC ManualControl
VAR_INPUT
	Switch: BOOL;
END_VAR
VAR
	ManualControl: BOOL;
	TimeForInterlockDelay: TIME := T#0.05S;
	ManualMode: BOOL;
	MotorSelection_1: MotorSelection;
	SelectedMotor: INT;
	temp: TIME;
	LowerLeftInterlock: TOF;
	LowerLeft: BOOL;
	LowerRightInterlock: TOF;
	LowerRight: BOOL;
END_VAR
VAR_OUTPUT
	Output: BOOL;
END_VAR
VAR // added by the converter: edge detectors and wires of the graphical bodies
    _w1, _w2, _w3, _w4, _w5, _w6, _w7, _w8, _w9, _w10, _w11 : BOOL;
    _rt1, _rt2, _rt3 : R_TRIG;
    _ft1, _ft2, _ft3 : F_TRIG;
END_VAR

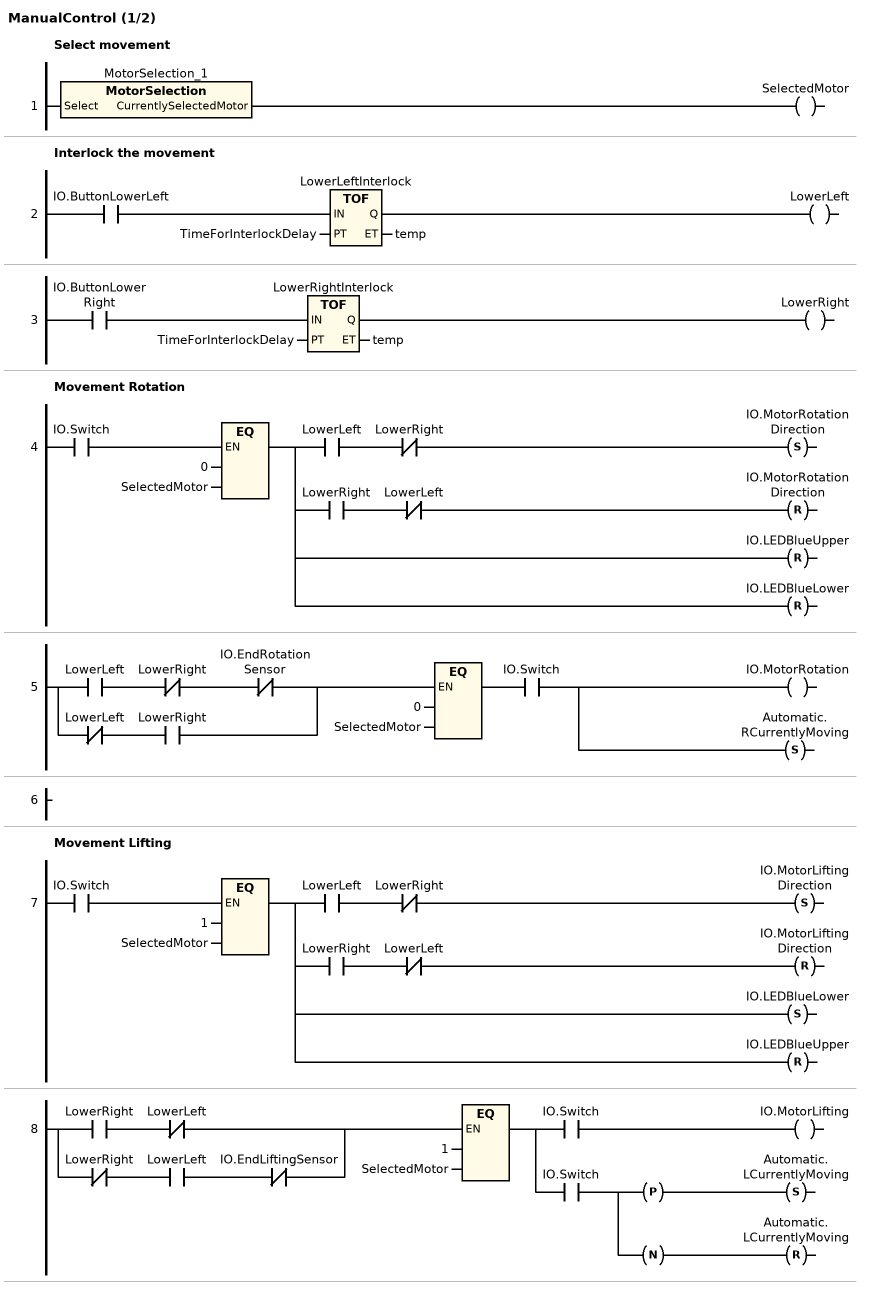
// NETWORK 1: Select movement
MotorSelection_1(Select := TRUE); // MotorSelection
SelectedMotor := MotorSelection_1.CurrentlySelectedMotor;

// NETWORK 2: Interlock the movement
LowerLeftInterlock(IN := IO.ButtonLowerLeft, PT := TimeForInterlockDelay, ET => temp); // TOF
LowerLeft := LowerLeftInterlock.Q;

// NETWORK 3
LowerRightInterlock(IN := IO.ButtonLowerRight, PT := TimeForInterlockDelay, ET => temp); // TOF
LowerRight := LowerRightInterlock.Q;

// NETWORK 4: Movement Rotation
_w1 := IO.Switch AND 0 = SelectedMotor;
IO.MotorRotationDirection S= _w1 AND LowerLeft AND NOT LowerRight;
IO.MotorRotationDirection R= _w1 AND LowerRight AND NOT LowerLeft;
IO.LEDBlueUpper R= _w1;
IO.LEDBlueLower R= _w1;

// NETWORK 5
_w2 := ((LowerLeft AND NOT LowerRight AND NOT IO.EndRotationSensor OR NOT LowerLeft AND LowerRight) AND 0 = SelectedMotor) AND IO.Switch;
IO.MotorRotation := _w2;
Automatic.RCurrentlyMoving S= _w2;

// NETWORK 6

// NETWORK 7: Movement Lifting
_w3 := IO.Switch AND 1 = SelectedMotor;
IO.MotorLiftingDirection S= _w3 AND LowerLeft AND NOT LowerRight;
IO.MotorLiftingDirection R= _w3 AND LowerRight AND NOT LowerLeft;
IO.LEDBlueLower S= _w3;
IO.LEDBlueUpper R= _w3;

// NETWORK 8
_w4 := (LowerRight AND NOT LowerLeft OR NOT LowerRight AND LowerLeft AND NOT IO.EndLiftingSensor) AND 1 = SelectedMotor;
IO.MotorLifting := _w4 AND IO.Switch;
_w5 := _w4 AND IO.Switch;
_rt1(CLK := _w5);
Automatic.LCurrentlyMoving S= _rt1.Q;
_ft1(CLK := _w5);
Automatic.LCurrentlyMoving R= _ft1.Q;

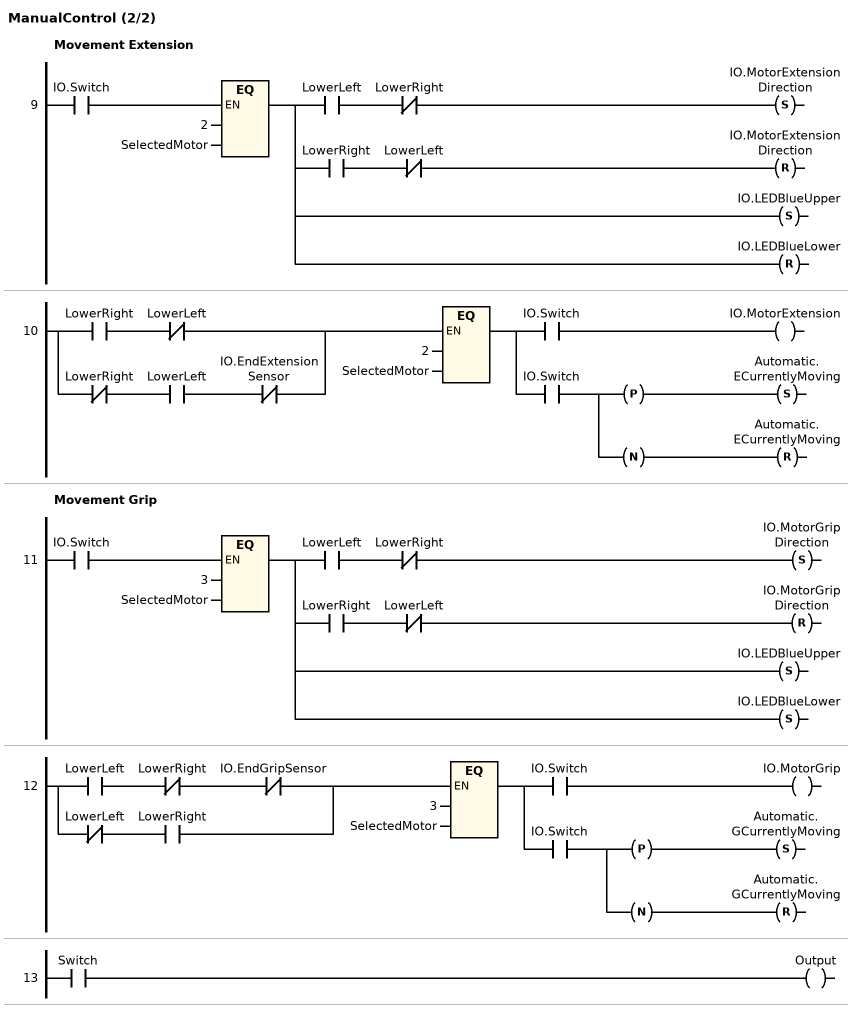
// NETWORK 9: Movement Extension
_w6 := IO.Switch AND 2 = SelectedMotor;
IO.MotorExtensionDirection S= _w6 AND LowerLeft AND NOT LowerRight;
IO.MotorExtensionDirection R= _w6 AND LowerRight AND NOT LowerLeft;
IO.LEDBlueUpper S= _w6;
IO.LEDBlueLower R= _w6;

// NETWORK 10
_w7 := (LowerRight AND NOT LowerLeft OR NOT LowerRight AND LowerLeft AND NOT IO.EndExtensionSensor) AND 2 = SelectedMotor;
IO.MotorExtension := _w7 AND IO.Switch;
_w8 := _w7 AND IO.Switch;
_rt2(CLK := _w8);
Automatic.ECurrentlyMoving S= _rt2.Q;
_ft2(CLK := _w8);
Automatic.ECurrentlyMoving R= _ft2.Q;

// NETWORK 11: Movement Grip
_w9 := IO.Switch AND 3 = SelectedMotor;
IO.MotorGripDirection S= _w9 AND LowerLeft AND NOT LowerRight;
IO.MotorGripDirection R= _w9 AND LowerRight AND NOT LowerLeft;
IO.LEDBlueUpper S= _w9;
IO.LEDBlueLower S= _w9;

// NETWORK 12
_w10 := (LowerLeft AND NOT LowerRight AND NOT IO.EndGripSensor OR NOT LowerLeft AND LowerRight) AND 3 = SelectedMotor;
IO.MotorGrip := _w10 AND IO.Switch;
_w11 := _w10 AND IO.Switch;
_rt3(CLK := _w11);
Automatic.GCurrentlyMoving S= _rt3.Q;
_ft3(CLK := _w11);
Automatic.GCurrentlyMoving R= _ft3.Q;

// NETWORK 13
Output := Switch;

END_FUNCTION_BLOCK

// ---- POUs/MotorSelection.TcPOU
FUNCTION_BLOCK PUBLIC MotorSelection
VAR_INPUT
	Select: BOOL;
END_VAR
VAR
	TimeForDelay: TIME := T#0.15S;
	MovementSelection: CTUD;
	SelectionCounter: CTUD := (LOAD := TRUE, PV := 3);
	ReachedMaxSelection: BOOL;
	ReachedMinSelection: BOOL;
	UpperLeftDelay: TOF;
	UpperRightDelay: TOF;
	tmnp: TIME;
	CU: BOOL;
	CD: BOOL;
	CUU: BOOL;
	CDD: BOOL;
	PositiveEdge1: R_TRIG;
	PositiveEdge2: R_TRIG;
	temporary: BOOL;
	CUU0: BOOL;
	CDD0: BOOL;
	temporary1: BOOL;
	BURpositiveEdge: BOOL;
	BULpositiveEdge: BOOL;
	temp2: BOOL;
	temp3: BOOL;
END_VAR
VAR_OUTPUT
	CurrentlySelectedMotor: WORD;
END_VAR
VAR // added by the converter: edge detectors and wires of the graphical bodies
    _rt1, _rt2, _rt3, _rt4 : R_TRIG;
END_VAR

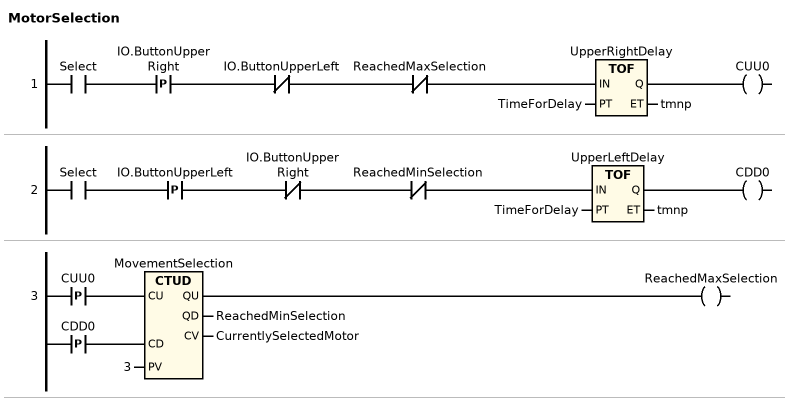
// NETWORK 1
_rt1(CLK := IO.ButtonUpperRight);
UpperRightDelay(
    IN := Select AND _rt1.Q AND NOT IO.ButtonUpperLeft AND NOT ReachedMaxSelection,
    PT := TimeForDelay,
    ET => tmnp); // TOF
CUU0 := UpperRightDelay.Q;

// NETWORK 2
_rt2(CLK := IO.ButtonUpperLeft);
UpperLeftDelay(
    IN := Select AND _rt2.Q AND NOT IO.ButtonUpperRight AND NOT ReachedMinSelection,
    PT := TimeForDelay,
    ET => tmnp); // TOF
CDD0 := UpperLeftDelay.Q;

// NETWORK 3
_rt3(CLK := CUU0);
_rt4(CLK := CDD0);
MovementSelection(
    CU := _rt3.Q,
    CD := _rt4.Q,
    PV := 3,
    QD => ReachedMinSelection,
    CV => CurrentlySelectedMotor); // CTUD
ReachedMaxSelection := MovementSelection.QU;

END_FUNCTION_BLOCK

// ---- POUs/MAIN.TcPOU
PROGRAM MAIN
VAR
	ManualControl_0: ManualControl;
	AutomaticControl_0: AutomaticControl;
END_VAR

// Initially it goes to position (0,0,0,0) and initializes motors by Initialize PRG.
// There is Safety PRG that keeps checking if motors are out of bounds.
// Motors are instantiated as global vars to retain their properties.
// CountCurrentPosition PRG is the only place where we count position using the sensors.
// RestorePreviousAutomaticState is a FB that gets execture cyclic until all the directions are set to previous positions.
// AutomaticControl FB remembers which recipe is being executed and recipe remembers its state.
VAR // added by the converter: edge detectors and wires of the graphical bodies
    _ft1 : F_TRIG;
    _rt1 : R_TRIG;
    _w1 : BOOL;
END_VAR

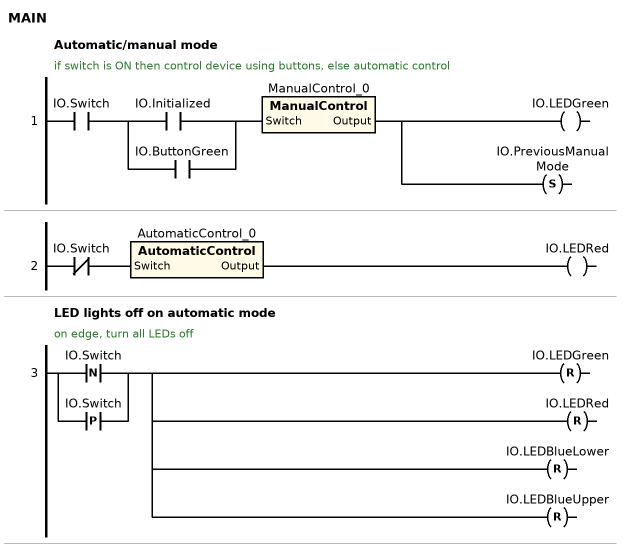
// NETWORK 1: Automatic/manual mode
// if switch is ON then control device using buttons, else automatic control
ManualControl_0(Switch := IO.Switch AND IO.Initialized OR IO.Switch AND IO.ButtonGreen); // ManualControl
IO.LEDGreen := ManualControl_0.Output;
IO.PreviousManualMode S= ManualControl_0.Output;

// NETWORK 2
AutomaticControl_0(Switch := NOT IO.Switch); // AutomaticControl
IO.LEDRed := AutomaticControl_0.Output;

// NETWORK 3: LED lights off on automatic mode
// on edge, turn all LEDs off
_ft1(CLK := IO.Switch);
_rt1(CLK := IO.Switch);
_w1 := _ft1.Q OR _rt1.Q;
IO.LEDGreen R= _w1;
IO.LEDRed R= _w1;
IO.LEDBlueLower R= _w1;
IO.LEDBlueUpper R= _w1;

END_PROGRAM

// ---- POUs/Recipe11.TcPOU
PROGRAM Recipe11
VAR_INPUT
	ExecutingRecipe1: BOOL;
END_VAR
VAR_OUTPUT
	SuccesfullyEnded: BOOL := FALSE;
END_VAR
VAR
	State: INT := 0;
	WoodInitialLiftingPosition: INT := 50;
	InitialExtensionPosition: INT := 388;
	MaxGripPosition: INT := 150;
	RotationDropOffPosition: INT := 300;
	PlasticsInitialLiftingPosition: INT := 250;
	PlasticsDropOffExtensionPosition: INT := 300;
	MetalInitialLiftingPosition: INT := 400;
	MetalDropOffExtensionPosition: INT := 500;
END_VAR

IF ExecutingRecipe1 THEN	// we start executing recipe1 (again)
	SuccesfullyEnded := FALSE;
END_IF

IF (NOT IO.Switch) AND (NOT SuccesfullyEnded) THEN
	IO.LEDGreen := 1;
	// WOOD:
	IF State = 0 THEN
		IF Automatic.LiftingPositionAuto < WoodInitialLiftingPosition THEN
			IO.MotorLiftingDirection := 0;
			IF (NOT Automatic.SafetyLON) THEN
				Automatic.LCurrentlyMoving := TRUE;
				IO.MotorLifting := 1;
			END_IF
		ELSE
			State := 1;
			IO.MotorLifting := 0;
			Automatic.LCurrentlyMoving := FALSE;
		END_IF
	ELSIF State = 1 THEN
		IF Automatic.ExtensionPositionAuto < InitialExtensionPosition THEN
			IO.MotorExtensionDirection := 0;
			IF NOT Automatic.SafetyEON THEN
				Automatic.ECurrentlyMoving := TRUE;
				IO.MotorExtension := 1;
			END_IF
		ELSE
			State := 2;
			IO.MotorExtension := 0;
			Automatic.ECurrentlyMoving := FALSE;
		END_IF
	ELSIF State = 2 THEN
		IF Automatic.GripPositionAuto < MaxGripPosition THEN
			IO.MotorGripDirection := 0;
			IF NOT Automatic.SafetyGON THEN
				Automatic.GCurrentlyMoving := TRUE;
				IO.MotorGrip := 1;
			END_IF
		ELSE
			State := 3;
			IO.MotorGrip := 0;
			Automatic.GCurrentlyMoving := FALSE;
		END_IF
	ELSIF State = 3 THEN
		IF NOT IO.EndLiftingSensor THEN
			IO.MotorLiftingDirection := 1;
			IF NOT Automatic.SafetyLON THEN
				Automatic.GCurrentlyMoving := TRUE;
				IO.MotorLifting := 1;
			END_IF
		ELSE
			State := 4;
			IO.MotorLifting := 0;
			Automatic.LCurrentlyMoving := FALSE;
		END_IF
	ELSIF State = 4 THEN
		IF Automatic.RotationPositionAuto < RotationDropOffPosition THEN
			IO.MotorRotationDirection := 0;
			IF NOT Automatic.SafetyRON THEN
				Automatic.RCurrentlyMoving := TRUE;
				IO.MotorRotation := 1;
			END_IF
		ELSE
			State := 5;
			IO.MotorRotation := 0;
			Automatic.RCurrentlyMoving := FALSE;
		END_IF
	ELSIF State = 5 THEN
		IF NOT IO.EndExtensionSensor THEN	// it drops wood in the nearest bin
			IO.MotorExtensionDirection := 1;
			IF NOT Automatic.SafetyEON THEN
				Automatic.ECurrentlyMoving := TRUE;
				IO.MotorExtension := 1;
			END_IF
		ELSE
			State := 6;
			IO.MotorExtension := 0;
			Automatic.ECurrentlyMoving := FALSE;
		END_IF
	ELSIF State = 6 THEN
		IF NOT IO.EndGripSensor THEN
			IO.MotorGripDirection := 1;
			IF NOT Automatic.SafetyGON THEN
				Automatic.GCurrentlyMoving := TRUE;
				IO.MotorGrip := 1;
			END_IF
		ELSE
			State := 7;
			IO.MotorGrip := 0;
			Automatic.GCurrentlyMoving := FALSE;
		END_IF
	ELSIF State = 7 THEN
		IF NOT IO.EndRotationSensor THEN
			IO.MotorRotationDirection := 1;
			IF NOT Automatic.SafetyRON THEN
				Automatic.RCurrentlyMoving := TRUE;
				IO.MotorRotation := 1;
			END_IF
		ELSE
			State := 8;
			IO.MotorRotation := 0;
			Automatic.RCurrentlyMoving := FALSE;
		END_IF
	END_IF
	
	// PLASTICS:
	IF State = 8 THEN
		IF Automatic.LiftingPositionAuto < PlasticsInitialLiftingPosition THEN
			IO.MotorLiftingDirection := 0;
			IF NOT Automatic.SafetyLON THEN
				Automatic.LCurrentlyMoving := TRUE;
				IO.MotorLifting := 1;
			END_IF
		ELSE
			State := 9;
			IO.MotorLifting := 0;
			Automatic.LCurrentlyMoving := FALSE;
		END_IF
	ELSIF State = 9 THEN
		IF Automatic.ExtensionPositionAuto < InitialExtensionPosition THEN
			IO.MotorExtensionDirection := 0;
			IF NOT Automatic.SafetyEON THEN
				Automatic.ECurrentlyMoving := TRUE;
				IO.MotorExtension := 1;
			END_IF
		ELSE
			State := 10;
			IO.MotorExtension := 0;
			Automatic.ECurrentlyMoving := FALSE;
		END_IF
	ELSIF State = 10 THEN
		IF Automatic.GripPositionAuto < MaxGripPosition THEN
			IO.MotorGripDirection := 0;
			IF NOT Automatic.SafetyGON THEN
				Automatic.GCurrentlyMoving := TRUE;
				IO.MotorGrip := 1;
			END_IF
		ELSE
			State := 11;
			IO.MotorGrip := 0;
			Automatic.GCurrentlyMoving := FALSE;
		END_IF
	ELSIF State = 11 THEN
		IF NOT IO.EndLiftingSensor THEN
			IO.MotorLiftingDirection := 1;
			IF NOT Automatic.SafetyLON THEN
				Automatic.LCurrentlyMoving := TRUE;
				IO.MotorLifting := 1;
			END_IF
		ELSE
			State := 12;
			IO.MotorLifting := 0;
			Automatic.LCurrentlyMoving := FALSE;
		END_IF
	ELSIF State = 12 THEN
		IF Automatic.RotationPositionAuto < RotationDropOffPosition THEN
			IO.MotorRotationDirection := 0;
			IF NOT Automatic.SafetyRON THEN
				Automatic.RCurrentlyMoving := TRUE;
				IO.MotorRotation := 1;
			END_IF
		ELSE
			State := 13;
			IO.MotorRotation := 0;
			Automatic.RCurrentlyMoving := FALSE;
		END_IF
	ELSIF State = 13 THEN
		IF Automatic.ExtensionPositionAuto > PlasticsDropOffExtensionPosition THEN	// it drops plastics into second nearest bin
			IO.MotorExtensionDirection := 1;
			IF NOT Automatic.SafetyEON THEN
				Automatic.ECurrentlyMoving := TRUE;
				IO.MotorExtension := 1;
			END_IF
		ELSE
			State := 14;
			IO.MotorExtension := 0;
			Automatic.ECurrentlyMoving := FALSE;
		END_IF
	ELSIF State = 14 THEN
		IF NOT IO.EndGripSensor THEN
			IO.MotorGripDirection := 1;
			IF NOT Automatic.SafetyGON THEN
				Automatic.GCurrentlyMoving := TRUE;
				IO.MotorGrip := 1;
			END_IF
		ELSE
			State := 15;
			IO.MotorGrip := 0;
			Automatic.GCurrentlyMoving := FALSE;
		END_IF
	ELSIF State = 15 THEN
		IF NOT IO.EndRotationSensor THEN
			IO.MotorRotationDirection := 0;
			IF NOT Automatic.SafetyRON THEN
				Automatic.RCurrentlyMoving := TRUE;
				IO.MotorRotation := 1;
			END_IF
		ELSE
			State := 16;
			IO.MotorRotation := 0;
			Automatic.RCurrentlyMoving := FALSE;
		END_IF
	END_IF
	
	// METAL:
	IF State = 16 THEN
		IF Automatic.LiftingPositionAuto < MetalInitialLiftingPosition THEN
			IO.MotorLiftingDirection := 0;
			IF NOT Automatic.SafetyLON THEN
				Automatic.LCurrentlyMoving := TRUE;
				IO.MotorLifting := 1;
			END_IF
		ELSE
			State := 17;
			IO.MotorLifting := 0;
			Automatic.LCurrentlyMoving := FALSE;
		END_IF
	ELSIF State = 17 THEN
		IF Automatic.ExtensionPositionAuto < InitialExtensionPosition THEN
			IO.MotorExtensionDirection := 0;
			IF NOT Automatic.SafetyEON THEN
				Automatic.ECurrentlyMoving := TRUE;
				IO.MotorExtension := 1;
			END_IF
		ELSE
			State := 18;
			IO.MotorExtension := 0;
			Automatic.ECurrentlyMoving := FALSE;
		END_IF
	ELSIF State = 18 THEN
		IF Automatic.GripPositionAuto < MaxGripPosition THEN
			IO.MotorGripDirection := 0;
			IF NOT Automatic.SafetyGON THEN
				Automatic.GCurrentlyMoving := TRUE;
				IO.MotorGrip := 1;
			END_IF
		ELSE
			State := 19;
			IO.MotorGrip := 0;
			Automatic.GCurrentlyMoving := FALSE;
		END_IF
	ELSIF State = 19 THEN
		IF NOT IO.EndLiftingSensor THEN
			IO.MotorLiftingDirection := 1;
			IF NOT Automatic.SafetyLON THEN
				Automatic.LCurrentlyMoving := TRUE;
				IO.MotorLifting := 1;
			END_IF
		ELSE
			State := 20;
			IO.MotorLifting := 0;
			Automatic.LCurrentlyMoving := FALSE;
		END_IF
	ELSIF State = 20 THEN
		IF Automatic.RotationPositionAuto < RotationDropOffPosition THEN
			IO.MotorRotationDirection := 0;
			IF NOT Automatic.SafetyRON THEN
				Automatic.RCurrentlyMoving := TRUE;
				IO.MotorRotation := 1;
			END_IF
		ELSE
			State := 21;
			IO.MotorRotation := 0;
			Automatic.RCurrentlyMoving := FALSE;
		END_IF
	ELSIF State = 21 THEN
		IF Automatic.ExtensionPositionAuto > MetalDropOffExtensionPosition THEN	// it drops metal into farthest bin
			IO.MotorExtensionDirection := 1;
			IF NOT Automatic.SafetyEON THEN
				Automatic.ECurrentlyMoving := TRUE;
				IO.MotorExtension := 1;
			END_IF
		ELSE
			State := 22;
			IO.MotorExtension := 0;
			Automatic.ECurrentlyMoving := FALSE;
		END_IF
	ELSIF State = 22 THEN
		IF NOT IO.EndGripSensor THEN
			IO.MotorGripDirection := 1;
			IF NOT Automatic.SafetyGON THEN
				Automatic.GCurrentlyMoving := TRUE;
				IO.MotorGrip := 1;
			END_IF
		ELSE
			State := 23;
			IO.MotorGrip := 0;
			Automatic.GCurrentlyMoving := FALSE;
		END_IF
	ELSIF State = 23 THEN
		IF NOT IO.EndRotationSensor THEN
			IO.MotorRotationDirection := 1;
			IF NOT Automatic.SafetyRON THEN
				Automatic.RCurrentlyMoving := TRUE;
				IO.MotorRotation := 1;
			END_IF
		ELSE
			State := 24;
			IO.MotorRotation := 0;
			Automatic.RCurrentlyMoving := FALSE;
		END_IF
	ELSIF State = 24 THEN
		SuccesfullyEnded := TRUE;
		State := 0;
		RETURN;
	END_IF
END_IF
RETURN;

END_PROGRAM
